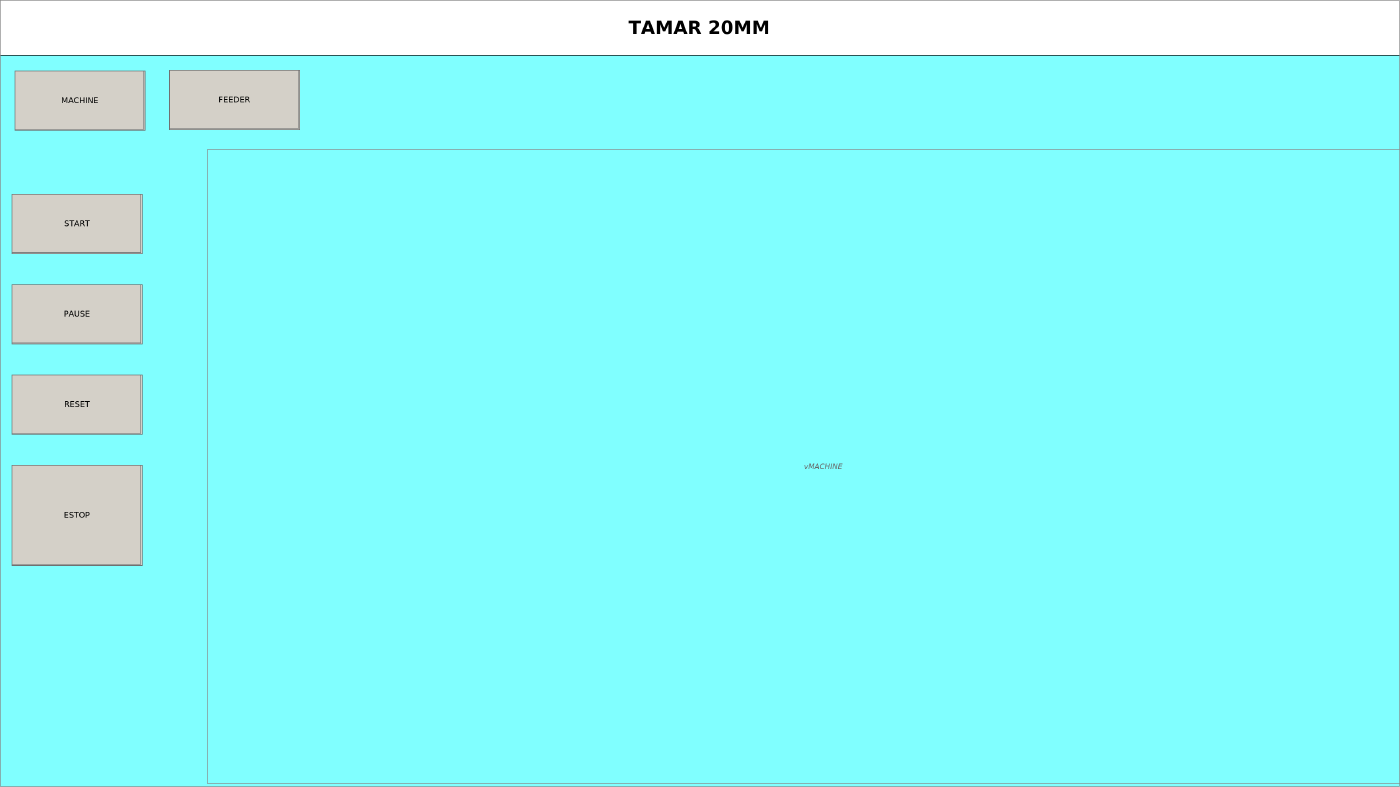
VISUALIZATION vCOMM  // 1920x1080
    Button (16,266 179x82), "START"
        OnMouseClick: FrameSelectionChange Selection=SelectedFrame=57b8a836-bac6-4cd4-9f68-9082885f5745, GlobSel=AssignType=Directly, SelType=Locally
    Rectangle (-3,-1 1924x77), "TAMAR 20MM"
    Button (16,390 179x82), "PAUSE"
        OnMouseClick: FrameSelectionChange Selection=SelectedFrame=57b8a836-bac6-4cd4-9f68-9082885f5745, GlobSel=AssignType=Directly, SelType=Locally
    Button (16,514 179x82), "RESET"
        OnMouseClick: FrameSelectionChange Selection=SelectedFrame=57b8a836-bac6-4cd4-9f68-9082885f5745, GlobSel=AssignType=Directly, SelType=Locally
    Button (16,638 179x138), "ESTOP"
        OnMouseClick: FrameSelectionChange Selection=SelectedFrame=57b8a836-bac6-4cd4-9f68-9082885f5745, GlobSel=AssignType=Directly, SelType=Locally
    Frame (284,205 1690x870)
        shows vMACHINE()
        shows vFEEDER(vFEEDER := fbFEEDER)
    Button (232,96 179x82), "FEEDER"
        OnMouseClick: FrameSelectionChange Selection=SelectedFrame=00e59953-e4a5-4fe1-b8af-e2191fac8d98, Selection=1, GlobSel=AssignType=Directly, SelType=Locally
    Button (20,97 179x82), "MACHINE"
        OnMouseClick: FrameSelectionChange Selection=SelectedFrame=00e59953-e4a5-4fe1-b8af-e2191fac8d98, GlobSel=AssignType=Directly, SelType=Locally
END_VISUALIZATION

(* stored: Version 1.1.0.1, ProductVersion 3.1.4024.12
   Visu vCOMM: Id {da002ba6-ee17-40f4-b476-8d87b46feaa7} *)
